// TIA Portal V20 export
DATA_BLOCK "SBK4"   // DB288
// stored: MemoryReserve 100
   VAR
      "X1-1 GATE EC STACK 2 NG BOX PB.LOCK" : Bool;
      "X2-1 GATE EC STACK 2 NG BOX PB.RESET" : Bool;
      "X3-1 DIFFERENTIAL PRESSURE SWITCH NC" : Bool;
      "X4-1 DIFFERENTIAL PRESSURE SWITCH 2 NC" : Bool;
      "X1-2 GATE EC STACK 2 NG BOX PB.UNLOCK" : Bool;
      "X2-2 SPARE" : Bool;
      "X3-2 DIFFERENTIAL PRESSURE SWITCH NO" : Bool;
      "X4-2 DIFFERENTIAL PRESSURE SWITCH 2 NO" : Bool;
   END_VAR
BEGIN
END_DATA_BLOCK
